Staubli VAL3: CustomPoll.pgx

public program CustomPoll()
  local num l_nNum
begin

  //引用位置:Kit:Poll.pgx
  //功能：用户在轮询函数中添加自己需要检查的内容
  // 可以添加报警信号
  //如果报警，则下电 dispower()
  //不需要加死循环，循环已经在poll.pgx中已经有了


  //  if dAlarm==true
  //    disablePower()
  //    logMsg("aAlarm 报警触发")
  //
  //  endIf






end
